FUNCTION_BLOCK Jack1Ctrl (* Basic Function Block Type *)
  (* Standard: 61499-2 *)
  (* Version 0.0, 3/23/2016, Aalto_IT, nxtControl GmbH, Template *)
  PACKAGE Main;
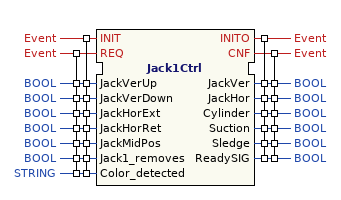
  EVENT_INPUT
    INIT WITH JackVerUp, JackVerDown, JackHorExt, JackHorRet, JackMidPos, Jack1_removes, Color_detected; (* Initialization Request *)
    REQ WITH JackVerUp, JackVerDown, JackHorExt, JackHorRet, JackMidPos, Jack1_removes, Color_detected; (* Normal Execution Request *)
  END_EVENT
  EVENT_OUTPUT
    INITO WITH JackVer, JackHor, Cylinder, Suction, Sledge, ReadySIG; (* Initialization Confirm *)
    CNF WITH JackVer, JackHor, Cylinder, Suction, Sledge, ReadySIG; (* Execution Confirmation *)
  END_EVENT
  VAR_INPUT
    JackVerUp : BOOL;
    JackVerDown : BOOL;
    JackHorExt : BOOL;
    JackHorRet : BOOL;
    JackMidPos : BOOL;
    Jack1_removes : BOOL;
    Color_detected : STRING;
  END_VAR
  VAR_OUTPUT
    JackVer : BOOL;
    JackHor : BOOL;
    Cylinder : BOOL;
    Suction : BOOL;
    Sledge : BOOL;
    ReadySIG : BOOL;
  END_VAR
  VAR
    TimeStamp : DATE_AND_TIME;
  END_VAR
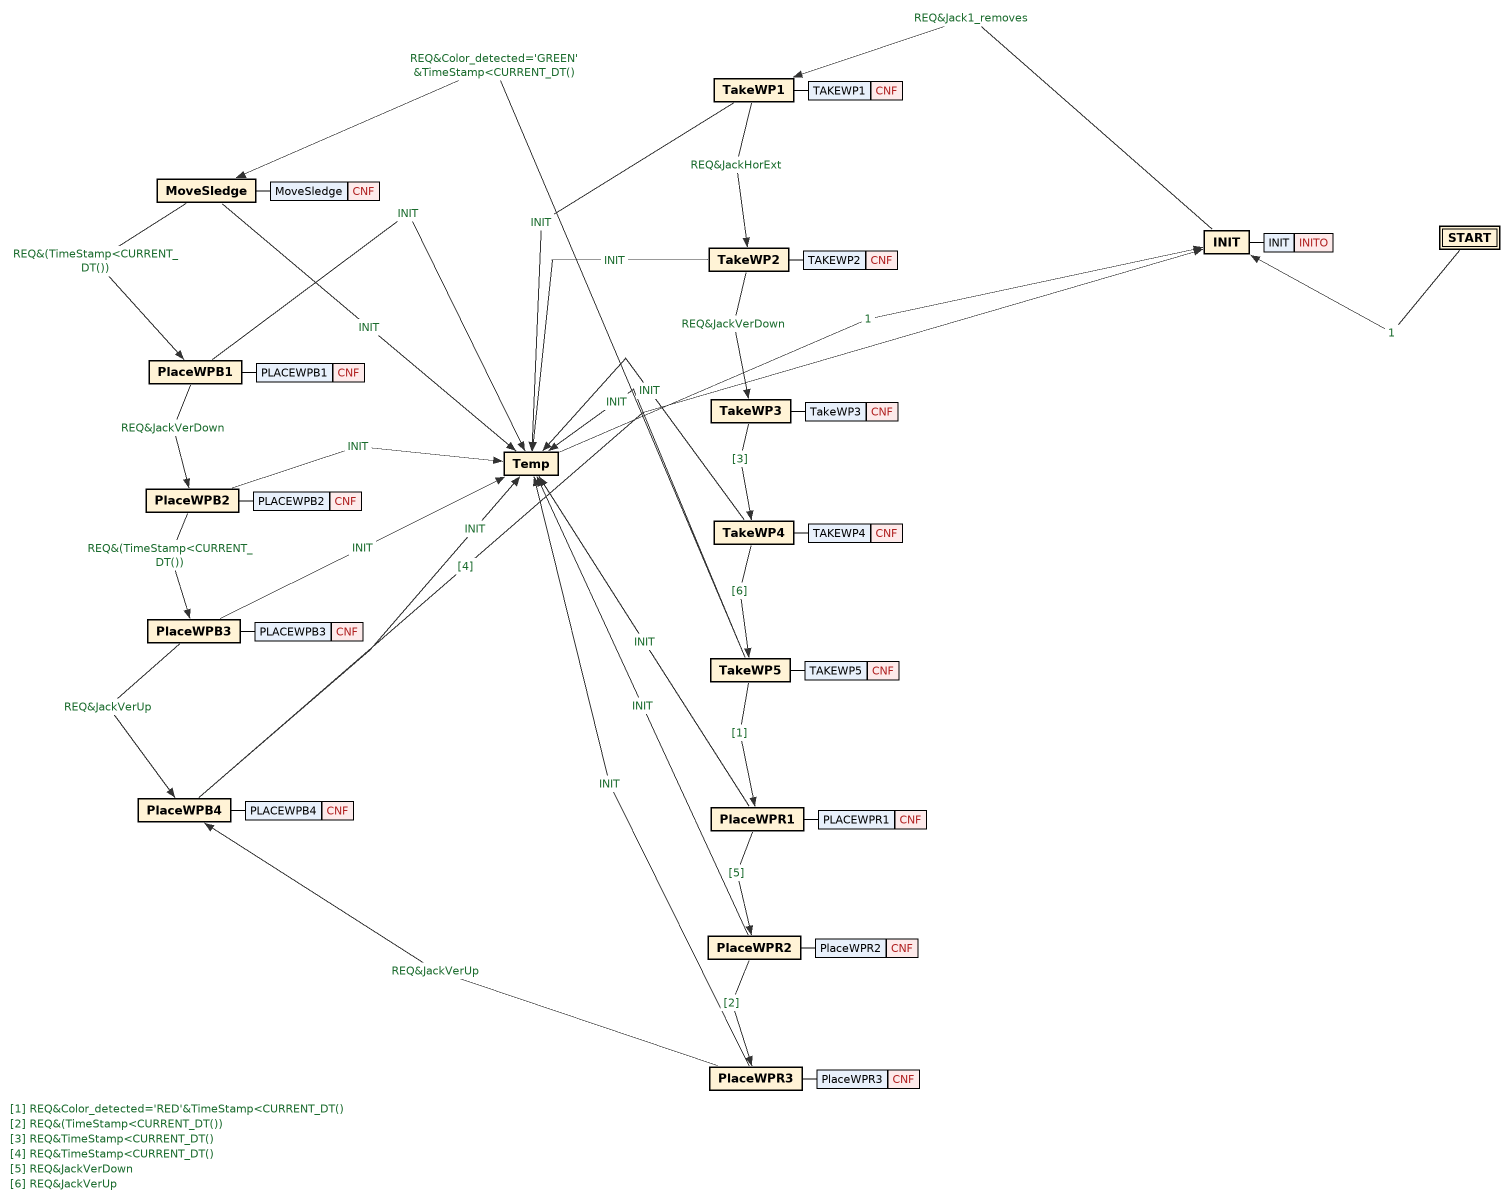
  EC_STATES
    START; (* Initial State *)
    INIT : INIT -> INITO; (* Initialization *)
    TakeWP1 : TAKEWP1 -> CNF;
    TakeWP2 : TAKEWP2 -> CNF;
    TakeWP4 : TAKEWP4 -> CNF;
    TakeWP5 : TAKEWP5 -> CNF;
    PlaceWPB1 : PLACEWPB1 -> CNF;
    MoveSledge : MoveSledge -> CNF;
    PlaceWPB2 : PLACEWPB2 -> CNF;
    PlaceWPB3 : PLACEWPB3 -> CNF;
    PlaceWPB4 : PLACEWPB4 -> CNF;
    PlaceWPR1 : PLACEWPR1 -> CNF;
    PlaceWPR2 : PlaceWPR2 -> CNF;
    PlaceWPR3 : PlaceWPR3 -> CNF;
    Temp;
    TakeWP3 : TakeWP3 -> CNF;
  END_STATES
  EC_TRANSITIONS
    START TO INIT := 1;
    TakeWP1 TO TakeWP2 := REQ&JackHorExt;
    TakeWP2 TO TakeWP3 := REQ&JackVerDown;
    TakeWP4 TO TakeWP5 := REQ&JackVerUp;
    MoveSledge TO PlaceWPB1 := REQ&(TimeStamp<CURRENT_DT());
    PlaceWPB1 TO PlaceWPB2 := REQ&JackVerDown;
    PlaceWPB2 TO PlaceWPB3 := REQ&(TimeStamp<CURRENT_DT());
    PlaceWPB3 TO PlaceWPB4 := REQ&JackVerUp;
    PlaceWPR2 TO PlaceWPR3 := REQ&(TimeStamp<CURRENT_DT());
    PlaceWPR3 TO PlaceWPB4 := REQ&JackVerUp;
    TakeWP1 TO Temp := INIT;
    TakeWP2 TO Temp := INIT;
    TakeWP4 TO Temp := INIT;
    TakeWP5 TO Temp := INIT;
    PlaceWPR1 TO Temp := INIT;
    PlaceWPR2 TO Temp := INIT;
    PlaceWPR3 TO Temp := INIT;
    MoveSledge TO Temp := INIT;
    PlaceWPB1 TO Temp := INIT;
    PlaceWPB2 TO Temp := INIT;
    PlaceWPB3 TO Temp := INIT;
    PlaceWPB4 TO Temp := INIT;
    Temp TO INIT := 1;
    TakeWP3 TO TakeWP4 := REQ&TimeStamp<CURRENT_DT();
    TakeWP5 TO PlaceWPR1 := REQ&Color_detected='RED'&TimeStamp<CURRENT_DT();
    PlaceWPR1 TO PlaceWPR2 := REQ&JackVerDown;
    TakeWP5 TO MoveSledge := REQ&Color_detected='GREEN'&TimeStamp<CURRENT_DT();
    INIT TO TakeWP1 := REQ&Jack1_removes;
    PlaceWPB4 TO INIT := REQ&TimeStamp<CURRENT_DT();
  END_TRANSITIONS
  ALGORITHM INIT IN ST: (* Initialization algorithm *)
JackVer:=0;
JackHor:=0;
Cylinder:=0;
Suction:=0;
Sledge:=0;
ReadySIG:=0;
  END_ALGORITHM
  ALGORITHM PLACEWPB1 IN ST: (* Suction on *)
;
JackVer:=1;
JackHor:=0;
Cylinder:=0;
Suction:=1;
Sledge:=1;
ReadySIG:=0;
  END_ALGORITHM
  ALGORITHM PLACEWPB2 IN ST:
;
JackVer:=1;
JackHor:=0;
Cylinder:=0;
Suction:=0;
Sledge:=1;
ReadySIG:=0;
TimeStamp:=ADD_DT_TIME(CURRENT_DT(),T#0.2s);
  END_ALGORITHM
  ALGORITHM PLACEWPB3 IN ST:
;
JackVer:=0;
JackHor:=0;
Cylinder:=0;
Suction:=0;
Sledge:=1;
ReadySIG:=0;
  END_ALGORITHM
  ALGORITHM PLACEWPB4 IN ST:
;
JackVer:=0;
JackHor:=0;
Cylinder:=0;
Suction:=0;
Sledge:=0;
ReadySIG:=1; // jack1 is done removing.
TimeStamp:=ADD_DT_TIME(CURRENT_DT(),T#0.5s);
  END_ALGORITHM
  ALGORITHM TAKEWP1 IN ST:
JackVer:=0;
JackHor:=1;
Cylinder:=0;
Suction:=0;
Sledge:=0;
ReadySIG:=0;
  END_ALGORITHM
  ALGORITHM TAKEWP2 IN ST:
JackVer:=1;
JackHor:=1;
Cylinder:=0;
Suction:=0;
Sledge:=0;
ReadySIG:=0;
  END_ALGORITHM
  ALGORITHM TAKEWP4 IN ST:
JackVer:=0;
JackHor:=1;
Cylinder:=0;
Suction:=1;
Sledge:=0;
ReadySIG:=0;
  END_ALGORITHM
  ALGORITHM TAKEWP5 IN ST:
JackVer:=0;
JackHor:=0;
Cylinder:=0;
Suction:=1;
Sledge:=0;
ReadySIG:=0;
TimeStamp := ADD_DT_TIME(CURRENT_DT(),T#2.0s);
  END_ALGORITHM
  ALGORITHM MoveSledge IN ST:
;
JackVer:=0;
JackHor:=0;
Cylinder:=0;
Suction:=1;
Sledge:=0;
ReadySIG:=0;
Sledge:=1; // Move Sledge to second position...
TimeStamp := ADD_DT_TIME(CURRENT_DT(),T#0.5s);
  END_ALGORITHM
  ALGORITHM PLACEWPR1 IN ST:
;
JackVer:=1;
JackHor:=0;
Cylinder:=0;
Suction:=1;
Sledge:=0;
ReadySIG:=0;
  END_ALGORITHM
  ALGORITHM PlaceWPR2 IN ST:
;
JackVer:=1;
JackHor:=0;
Cylinder:=0;
Suction:=0;
Sledge:=0;
ReadySIG:=0;
TimeStamp:=ADD_DT_TIME(CURRENT_DT(),T#0.2s);
  END_ALGORITHM
  ALGORITHM PlaceWPR3 IN ST:
;
JackVer:=0;
JackHor:=0;
Cylinder:=0;
Suction:=0;
Sledge:=0;
ReadySIG:=0;
  END_ALGORITHM
  ALGORITHM PlaceWPR4 IN ST:
;
JackVer:=0;
JackHor:=0;
Cylinder:=0;
Suction:=0;
Sledge:=0;
ReadySIG:=0;
  END_ALGORITHM
  ALGORITHM TakeWP3 IN ST:
;
JackVer:=1;
JackHor:=1;
Cylinder:=0;
Suction:=1;
Sledge:=0;
ReadySIG:=0;
TimeStamp := ADD_DT_TIME(CURRENT_DT(),T#0.3s);
  END_ALGORITHM
END_FUNCTION_BLOCK
